(* PLC project SafeLOGIC-1, BrAutomation SafeDESIGNER  4.3.4.4 *)
(* stored: companyURL http://www.br-automation.com, creationDateTime Thu Jun 24 15:07:09 2021 *)

PROGRAM Main

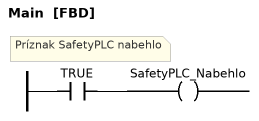
(* FBD diagram, written out as Structured Text *)
(* Príznak SafetyPLC nabehlo *)
SafetyPLC_Nabehlo := TRUE;
END_PROGRAM
